{attribute 'qualified_only'}
{attribute 'strict'}
TYPE E_SlideNest_State :
(
	//GENERIC
	ABORTED				,
	HOMING				,
	READY				,
	MANUAL_MODE			,
	STOPPING			,
	//SPECIFIC FOR EVERY STATION
	MOVE_RIGHT			,
	MOVE_LEFT			,
	DONE				,
	RESET				
);
END_TYPE

(* stored: Version 1.1.0.1, ProductVersion 3.1.4026.18
   DUT E_SlideNest_State: Id {bebd36fe-a8e0-4ba4-a698-4f514c6128fc} *)
